Staubli VAL3: start.pgx

public program start()
begin
  // end of cycle
  cycleStatus:bToEnd=true
  watch(cycleStatus:bToEnd==false,1)
end
